PROGRAM Student
VAR
	minVal: INT := 1; 
	maxVal: INT := 100;
	Roll4Motivation: DRAND;
	RandomReal: REAL;
	Moti: INT;
	StartWorking: SR;
	StudentNotification: BOOL;
	DontWantTo: BOOL;
	RisingSun: R_TRIG;
	RSun: BOOL;
END_VAR

//set notification
StartWorking(SET1:=GVL.StartPls , RESET:=GVL.Finished OR DontWantTo , Q1=>StudentNotification );

//daily rising edge signal
RisingSun(CLK:=GVL.Cycle , Q=>RSun );

//daily motivation amount
IF RSun = TRUE THEN
	Roll4Motivation(Seed:= , Num=>RandomReal );
	Moti := minVal + REAL_TO_INT(RandomReal * (maxVal - minVal + 1));
END_IF

//when the student has a notification pending they will decide what to do with it depending on the amount of motivation they have that given day
IF StudentNotification = TRUE THEN
	IF (GVL.MainDueIn*-1) + Moti > 69 THEN
		GVL.Finished := TRUE;
	ELSIF (GVL.MainDueIn*-1) + Moti < 69 THEN
		DontWantTo := TRUE;
	END_IF
END_IF

END_PROGRAM

(* stored: Version 1.1.0.1, ProductVersion 3.1.4024.12
   POU Student: Id {f7fde937-a145-4461-be69-639376c0a1a8}, SpecialFunc None *)
